(* PLC project Unnamed, Unknown Unnamed 1 *)
(* stored: creationDateTime 2024-10-19T20:32:53, modificationDateTime 2024-10-25T17:35:29 *)

(* Manipular un LED según la iluminación detectada por un LDR *)
PROGRAM program0
  VAR
    red AT %QX0.2 : BOOL := 0;  (* Controla el color rojo del LED. *)
    green AT %QX0.3 : BOOL := 0;  (* Controla el color verde del LED. *)
    blue AT %QX0.4 : BOOL := 0;  (* Controla el color azul del LED. *)
    light_sensor AT %IW0 : INT;  (* Nivel de iluminación medido por el LDR. *)
  END_VAR
  VAR
    light_threshold : INT := 450;  (* Nivel mínimo de Iluminación aceptable. *)
  END_VAR
  VAR
    correct_pin AT %IX0.6 : BOOL;  (* Botón de PIN correcto presionado. *)
    incorrect_pin AT %IX0.7 : BOOL;  (* Botón de PIN incorrecto presionado. *)
  END_VAR
  VAR
    max_failed_attempts : INT := 3;  (* Total de intentos fallidos permitidos. *)
    open : BOOL := 0;  (* Verdadero cuando el candado está abierto. *)
    closed : BOOL := 1;  (* Verdadero cuando el candado está cerrado. *)
    alarmed : BOOL := 0;  (* Verdadero cuando el candado está alarmado. *)
    disabled : BOOL := 0;  (* Verdadero cuando hay suficiente iluminación. *)
    FAILED_ATTEMPT_BLINK : TP;
    ALARM_BLINK : TP;
    ALARM_BLINK_TOGGLER : TOF;
    ALARM_TIMER : TON;
    FAILED_ATTEMPTS_COUNTER : CTU;
    BLUE_TO_RED_TRIGGER : R_TRIG;
    RED_TO_BLUE_TRIGGER : F_TRIG;
    STOP_BLINK_TRIGGER : F_TRIG;
    ENABLE_TRIGGER : F_TRIG;
    DISABLE_TRIGGER : R_TRIG;
  END_VAR
  VAR  (* added by the conversion: wires and edge detectors of the diagram *)
    R_TRIG1 : R_TRIG;
    R_TRIG2 : R_TRIG;
    R_TRIG3 : R_TRIG;
    R_TRIG4 : R_TRIG;
    F_TRIG5 : F_TRIG;
    _GE88_OUT : BOOL;
    R_TRIG6 : R_TRIG;
    F_TRIG7 : F_TRIG;
  END_VAR

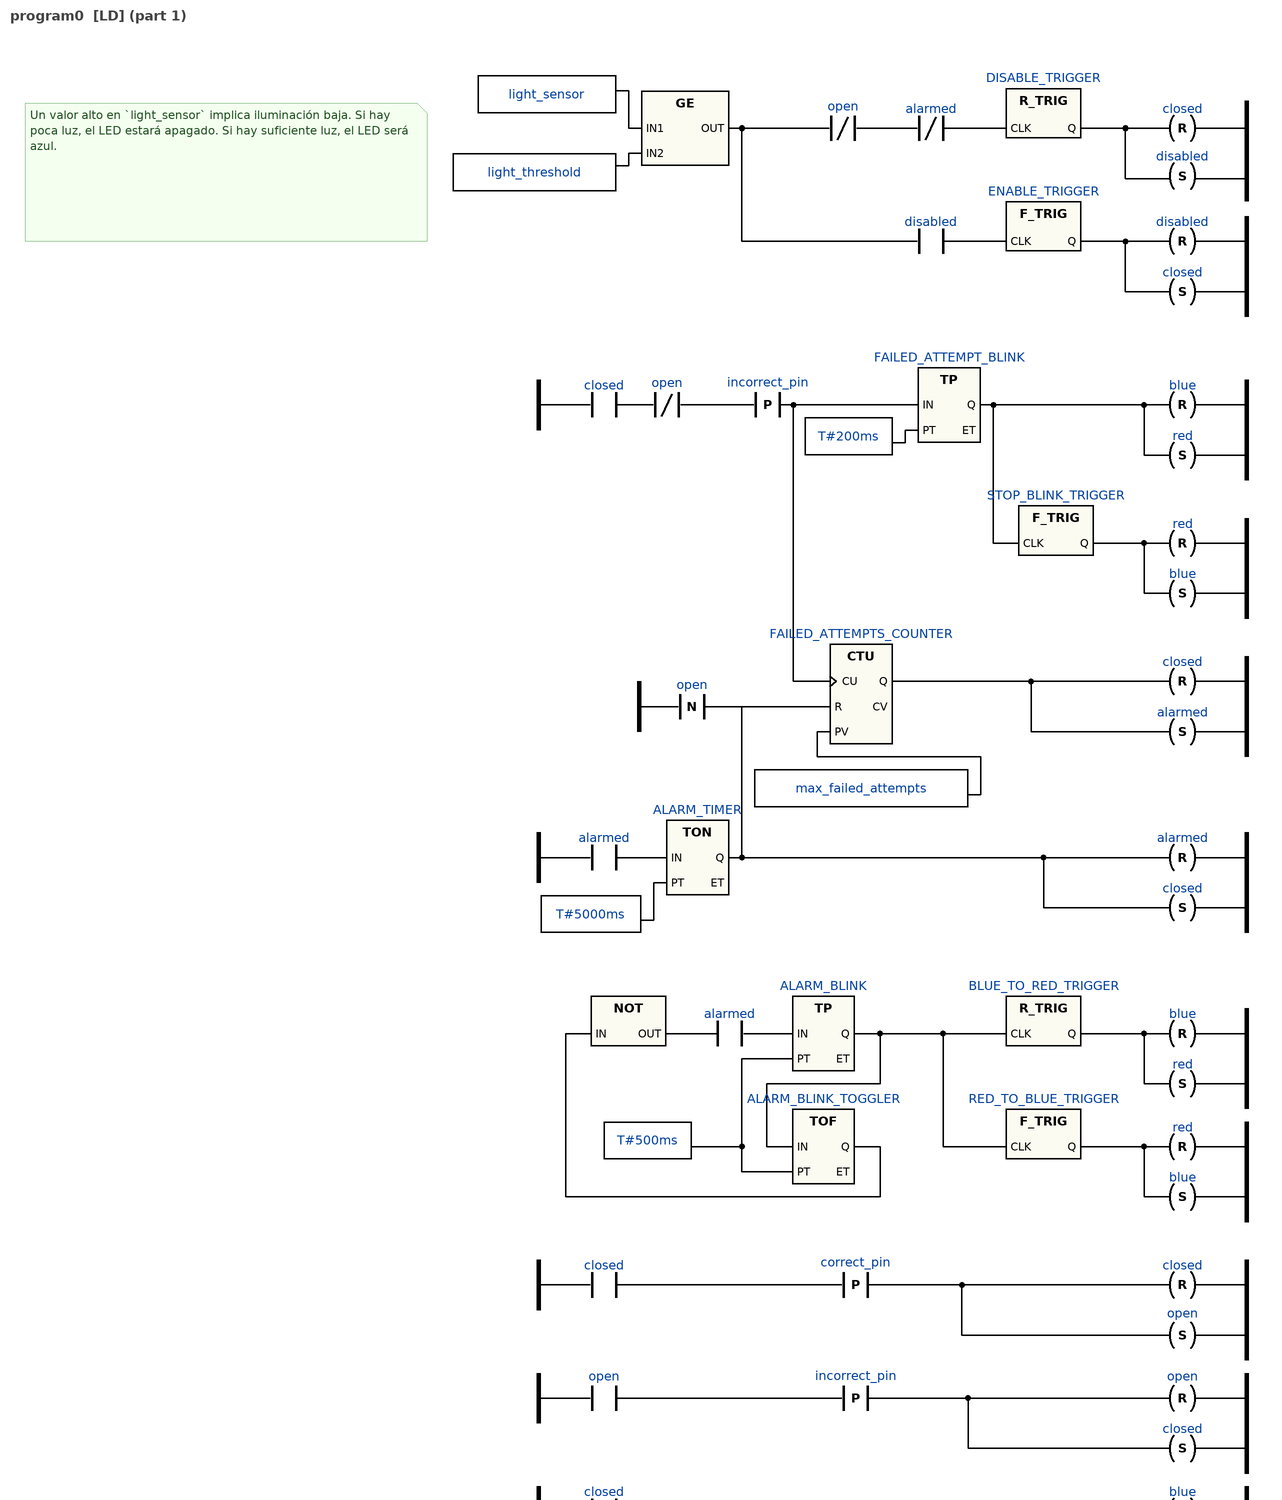
(* LD diagram, written out as Structured Text *)
(* Un valor alto en `light_sensor` implica iluminación baja. Si hay poca luz, el LED estará apagado. Si hay suficiente luz, el LED será azul. *)
R_TRIG1(CLK := correct_pin);
IF closed AND R_TRIG1.Q THEN open := TRUE; END_IF;
R_TRIG2(CLK := incorrect_pin);
IF open AND R_TRIG2.Q THEN closed := TRUE; END_IF;
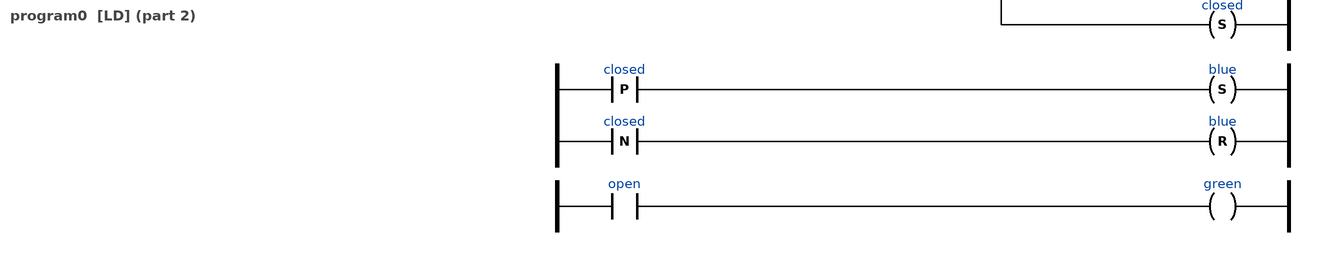
green := open;
R_TRIG3(CLK := incorrect_pin);
FAILED_ATTEMPT_BLINK(IN := closed AND NOT open AND R_TRIG3.Q, PT := T#200ms);
IF FAILED_ATTEMPT_BLINK.Q THEN blue := FALSE; END_IF;
IF FAILED_ATTEMPT_BLINK.Q THEN red := TRUE; END_IF;
IF closed AND R_TRIG1.Q THEN closed := FALSE; END_IF;
IF open AND R_TRIG2.Q THEN open := FALSE; END_IF;
R_TRIG4(CLK := closed AND NOT open AND R_TRIG3.Q);
ALARM_TIMER(IN := alarmed, PT := T#5000ms);
F_TRIG5(CLK := open);
FAILED_ATTEMPTS_COUNTER(CU := R_TRIG4.Q, R := ALARM_TIMER.Q OR F_TRIG5.Q, PV := max_failed_attempts);
IF FAILED_ATTEMPTS_COUNTER.Q THEN alarmed := TRUE; END_IF;
ALARM_BLINK_TOGGLER(IN := ALARM_BLINK.Q, PT := T#500ms);
ALARM_BLINK(IN := NOT ALARM_BLINK_TOGGLER.Q AND alarmed, PT := T#500ms);
BLUE_TO_RED_TRIGGER(CLK := ALARM_BLINK.Q);
IF BLUE_TO_RED_TRIGGER.Q THEN blue := FALSE; END_IF;
IF BLUE_TO_RED_TRIGGER.Q THEN red := TRUE; END_IF;
IF ALARM_TIMER.Q THEN alarmed := FALSE; END_IF;
IF ALARM_TIMER.Q THEN closed := TRUE; END_IF;
IF FAILED_ATTEMPTS_COUNTER.Q THEN closed := FALSE; END_IF;
RED_TO_BLUE_TRIGGER(CLK := ALARM_BLINK.Q);
IF RED_TO_BLUE_TRIGGER.Q THEN red := FALSE; END_IF;
IF RED_TO_BLUE_TRIGGER.Q THEN blue := TRUE; END_IF;
STOP_BLINK_TRIGGER(CLK := FAILED_ATTEMPT_BLINK.Q);
IF STOP_BLINK_TRIGGER.Q THEN red := FALSE; END_IF;
IF STOP_BLINK_TRIGGER.Q THEN blue := TRUE; END_IF;
_GE88_OUT := light_sensor >= light_threshold;
DISABLE_TRIGGER(CLK := _GE88_OUT AND NOT open AND NOT alarmed);
IF DISABLE_TRIGGER.Q THEN closed := FALSE; END_IF;
IF DISABLE_TRIGGER.Q THEN disabled := TRUE; END_IF;
ENABLE_TRIGGER(CLK := _GE88_OUT AND disabled);
IF ENABLE_TRIGGER.Q THEN disabled := FALSE; END_IF;
IF ENABLE_TRIGGER.Q THEN closed := TRUE; END_IF;
R_TRIG6(CLK := closed);
IF R_TRIG6.Q THEN blue := TRUE; END_IF;
F_TRIG7(CLK := closed);
IF F_TRIG7.Q THEN blue := FALSE; END_IF;
END_PROGRAM

CONFIGURATION Config0
  RESOURCE Res0 ON PLC
    TASK task0(INTERVAL := T#20ms, PRIORITY := 0);
    PROGRAM instance0 WITH task0 : program0;
  END_RESOURCE
END_CONFIGURATION
